(* CODESYS project retain.paras.190613.2.project

Project tree, tasks and I/O mapping:
  MIC7001 : Changsha Xiangji-ARM Cortex A9(xilinx zynq7000)-linux, Changsha Xiangji Hiden Technology Co.Ltd, version 3.5.10.40
    application Application
      libraries: Standard, * (System); CAA File, * (CAA Technical Workgroup); CAA Types Extern, * (CAA Technical Workgroup); CAA Callback Extern, * (CAA Technical Workgroup); SysMem, * (System); Util, 3.5.11.0 (System); SysFile, 3.5.9.0 (System); SysTypes Interfaces, * (System); CAN API, 1.0.0.3 (3S - Smart Software Solutions GmbH); SysTime, * (System); CAA DTUtil Extern, 3.5.12.0 (CAA Technical Workgroup); CAA SerialCom, 3.5.12.0 (CAA Technical Workgroup); cyber gpio, 3.5.10.40 (cyber); AC_DataLog, 3.5.13.0 (3S - Smart Software Solutions GmbH)
      task MainTask (cyclic, interval 20 ms, priority 15) calls prg_main
      task task_retain (cyclic, interval 200 ms, priority 19) calls prg_retain_paras
      global variables GVL
      retain_para/
        data type DUT_PARA_DINT
        data type DUT_PARA_REAL
        function block FB_PARA_DINT [ST]: wr_all, clear_all, rd_all, chk_chg
        function block FB_PARA_REAL [ST]: clear_all, wr_all, rd_all, chk_chg
        program prg_retain_paras [ST]
      program prg_main [ST]
    SoftMotion General Axis Pool
  text list GlobalTextList
*)

// MIC7001/Application/retain_para/DUT_PARA_DINT
TYPE DUT_PARA_DINT :
STRUCT
	num:UINT := 64;  //可根据需要设置总数量，最后一个为校验和，不可用
	para:ARRAY[0..64] OF DINT;  //三行中的总数量需要严格一致,位置0 用于存放魔法数字
	old_val:ARRAY[0..64] OF DINT; //三行中的总数量需要严格一致,位置0 用于存放魔法数字
	filename :STRING := '/userapp/mic_dint.txt';  
END_STRUCT
END_TYPE

// MIC7001/Application/retain_para/DUT_PARA_REAL
TYPE DUT_PARA_REAL :
STRUCT
	num:UINT := 256; //可根据需要设置总数量，最后一个为校验和，不可用
	para:ARRAY[0..256] OF REAL;  //三行中的总数量需要严格一致,位置0 用于存放魔法数字
	old_val:ARRAY[0..256] OF REAL; //三行中的总数量需要严格一致,位置0 用于存放魔法数字
	filename :STRING := '/userapp/mic_real.txt';  
END_STRUCT
END_TYPE

// MIC7001/Application/GVL
VAR_GLOBAL
	user_para_01: DINT := 1234;
	user_para_02: DINT := 3323;
	user_para_03: DINT := 4322;
END_VAR

// MIC7001/Application/prg_main
PROGRAM prg_main
VAR
	cntr :dint := 0;
END_VAR


cntr := cntr + 1;

IF cntr > 100 THEN
	gvl.user_para_01 := gvl.user_para_01 + 1;
	gvl.user_para_02 := gvl.user_para_02 + 2;
	
	gvl.user_para_03 := gvl.user_para_03 + 0;
	
	cntr := 0;
END_IF

END_PROGRAM

// MIC7001/Application/retain_para/prg_retain_paras
PROGRAM prg_retain_paras
VAR
	data_stat:UINT := 0;
    myRetainMigicNumber:DINT := 1324904337;  //本机型的魔法数字，必须修改，越随机越好
END_VAR

VAR_INPUT
	para_dint:DUT_PARA_DINT;
	retain_dint:FB_PARA_DINT;
END_VAR

//整数参数掉电存储例程

// (1) 拷贝本工程内的 parameters 目录到用户自己的工程;
// (2) 将其中的prg_retain_paras 程序拷贝到 某一个任务中；
// (3) 使用自己定义的变量替换掉 gvl.user_para_01,   gvl.user_para_02 和 gvl.user_para_03, 并更改本程序中对应的变量
// (4) 如果需要保存更多的变量，可仿照本例增加变量（默认支持64个） 

retain_dint(enable := TRUE, pPara := ADR(para_dint));

CASE data_stat OF
0:
	IF retain_dint.zero OR para_dint.para[0] <> myRetainMigicNumber  THEN   //数据为空或者魔法数字错误，恢复初始值
		para_dint.para[0] := myRetainMigicNumber;
		para_dint.para[1] := gvl.user_para_01;
		para_dint.para[2] := gvl.user_para_02;
		para_dint.para[3] := gvl.user_para_03;
		//para_dint.para[4] := gvl.user_para_04;  
		//可在此处添加新的用户变量
	ELSE
		gvl.user_para_01 := para_dint.para[1];
		gvl.user_para_02 := para_dint.para[2];
		gvl.user_para_03 := para_dint.para[3];
		//gvl.user_para_04 := para_dint.para[4];  
		//可在此处添加新的用户变量
		
		data_stat := 10;
	END_IF
10:
	para_dint.para[1] := gvl.user_para_01;
	para_dint.para[2] := gvl.user_para_02;
	para_dint.para[3] := gvl.user_para_03;
	//para_dint.para[4] := gvl.user_para_04;  
	//可在此处添加新的用户变量
	
END_CASE

END_PROGRAM

// MIC7001/Application/retain_para/FB_PARA_DINT
FUNCTION_BLOCK FB_PARA_DINT
VAR_INPUT
	enable:BOOL := FALSE;
	clear:BOOL := FALSE;
	pPara:POINTER TO DUT_PARA_DINT;
END_VAR

VAR_OUTPUT
	ok:BOOL := FALSE;
	zero:BOOL := FALSE;
END_VAR

VAR
	hFile: RTS_IEC_HANDLE := 0;
	sync:BOOL := FALSE;  
	stat:UINT:= 0;
	
	i :UINT;
END_VAR


IF NOT enable OR pPara^.num < 1 THEN
	stat := 0;
	RETURN;
END_IF

CASE stat OF
	0:  //init
		IF rd_all(pPara^.filename)	THEN 
			zero := FALSE;
			ok := TRUE;
			stat := 10;
		ELSE
			clear_all();
			IF wr_all(pPara^.filename) THEN
				zero := TRUE;
				ok := FALSE;
				stat := 10;
			END_IF
		END_IF
	
	10: // normal
		IF chk_chg() THEN
			ok := FALSE;
			IF wr_all(pPara^.filename) THEN
				ok := TRUE;
				zero := FALSE;
			END_IF
		END_IF	
		
		IF clear THEN
			clear_all();
			IF wr_all(pPara^.filename) THEN
				zero := TRUE;
				ok := FALSE;
			END_IF
		END_IF
END_CASE

METHOD wr_all : bool
VAR_INPUT
	filename:STRING(256);
END_VAR

VAR
	iNumber:INT;
	udiByteWrite:LWORD;
	udiPos:UDINT;
	udiOpenError: RTS_IEC_RESULT;
	udiWriteError: RTS_IEC_RESULT;
	str_size:DWORD;
	str: STRING(255);
	check_sum: DINT;
END_VAR
wr_all := FALSE;
hFile := sysfileopen(szFile := filename, am := sysfile.AM_WRITE, pResult := ADR(udiOpenError));
IF hFile = RTS_INVALID_HANDLE THEN
	RETURN;
END_IF

udiPos := SysFileSetPos(hFile:=hFile, ulOffset := 0);

check_sum := 0;
str:= ANY_TO_STRING('');
FOR i := 0 TO pPara^.num DO
	IF i = pPara^.num THEN  //the last val, check_sum
		pPara^.para[i] := check_sum;
	ELSE
		check_sum := check_sum + pPara^.para[i];
	END_IF
	str := concat(str, ANY_TO_STRING(pPara^.para[i]));
	str := concat(str, ANY_TO_STRING('$N'));
	str_size := ANY_TO_DWORD(len(str));
	IF str_size > 200 THEN
		udiByteWrite := sysfile.SysFileWrite(hFile := hFile,pbyBuffer := ADR(str),ulSize := str_size, pResult := ADR(udiWriteError));
		IF udiByteWrite = str_size THEN
			str := '';
		END_IF
	END_IF	
END_FOR
udiByteWrite := sysfile.SysFileWrite(hFile := hFile,pbyBuffer := ADR(str),ulSize := str_size, pResult := ADR(udiWriteError));
	
IF udiByteWrite <> str_size THEN
	sysfile.SysFileClose(hFile);
	RETURN;
END_IF
sysfile.SysFileClose(hFile);

	
FOR i := 0 TO pPara^.num DO
	pPara^.old_val[i] := pPara^.para[i];
END_FOR

hFile := 0;

wr_all := TRUE;
END_METHOD

METHOD clear_all : bool
VAR_INPUT
	
END_VAR
FOR i := 0 TO pPara^.num DO
	pPara^.para[i] := 0;
	pPara^.old_val[i] := 0;
END_FOR

clear_all := TRUE;
END_METHOD

METHOD rd_all : bool
VAR_INPUT
	filename:STRING(256);
END_VAR

VAR
	iNumber:INT;
	udiByteRead:LWORD;
	udiPos:UDINT;
	udiOpenError: RTS_IEC_RESULT;
	udiReadError: RTS_IEC_RESULT;
	str: STRING(255);
	ulOffset:DWORD;
	batch: BOOL;
	check_sum: DINT;
END_VAR
rd_all := FALSE;

hFile := sysfileopen(szFile := filename, am := sysfile.AM_READ, pResult:= ADR(udiOpenError));
IF hFile = RTS_INVALID_HANDLE THEN
	RETURN;
END_IF

ulOffset := 0;
batch := TRUE;

check_sum := 0;
FOR i := 0 TO pPara^.num DO
	IF udiByteRead < 50 AND batch THEN
		udiPos := SysFileSetPos(hFile:=hFile, ulOffset := ulOffset);
		udiByteRead := sysfile.SysFileRead(hfile := hFile,pbyBuffer := ADR(str), ulSize := 255 , pResult := ADR(udiReadError));
		IF udiByteRead < 255 THEN
			batch := FALSE;
		END_IF
	END_IF
	IF udiByteRead < 1 THEN  //读取失败
		sysfile.SysFileClose(hFile := hFile);
		RETURN;
	END_IF

	iNumber := find(str, '$N');
	IF iNumber < 2 THEN
		sysfile.SysFileClose(hFile := hFile);
		RETURN;
	END_IF
	
	pPara^.para[i] := STRING_TO_DINT(left(str,iNumber-1));
	str := delete(str, iNumber,1);
	pPara^.old_val[i] := pPara^.para[i];
	
	udiByteRead := udiByteRead - ANY_TO_LWORD(iNumber);
	ulOffset := ulOffset + ANY_TO_DWORD(iNumber);

	IF i = pPara^.num THEN
		IF check_sum <> pPara^.para[i] THEN
			RETURN;  //error
		END_IF
	ELSE
		check_sum := check_sum + pPara^.para[i];
	END_IF
END_FOR

sysfile.SysFileClose(hFile := hFile);
rd_all := TRUE;
END_METHOD

METHOD chk_chg : bool
VAR_INPUT
END_VAR

VAR
	i :UINT;
END_VAR
chk_chg := TRUE;

FOR i := 0 TO pPara^.num  DO
	IF pPara^.para[i] <> pPara^.old_val[i] THEN
		RETURN;
	END_IF
END_FOR

chk_chg := FALSE;
END_METHOD

END_FUNCTION_BLOCK

// MIC7001/Application/retain_para/FB_PARA_REAL
FUNCTION_BLOCK FB_PARA_REAL
VAR_INPUT
	enable:BOOL := FALSE;
	clear:BOOL := FALSE;
	pPara:POINTER TO DUT_PARA_REAL;
END_VAR

VAR_OUTPUT
	ok:BOOL := FALSE;
	zero:BOOL := FALSE;
END_VAR

VAR
	hFile: RTS_IEC_HANDLE := 0;
	sync:BOOL := FALSE;  
	stat:UINT:= 0;
	
	i :UINT;
	str:STRING(1024);
END_VAR


IF NOT enable OR pPara^.num < 1 THEN
	stat := 0;
	RETURN;
END_IF

CASE stat OF
	0:  //init
		IF rd_all(pPara^.filename)	THEN 
			zero := FALSE;
			stat := 10;
		ELSE
			clear_all();
			IF wr_all(pPara^.filename) THEN
				zero := TRUE;
				stat := 10;
			END_IF
		END_IF
	
	10: // normal
		IF chk_chg() THEN
			ok := FALSE;
			IF wr_all(pPara^.filename) THEN
				ok := TRUE;
				zero := FALSE;
			END_IF
		END_IF	
		
		IF clear THEN
			clear_all();
			IF wr_all(pPara^.filename) THEN
				zero := TRUE;
			END_IF
		END_IF
END_CASE

METHOD clear_all : bool
VAR_INPUT
	
END_VAR
FOR i := 0 TO pPara^.num DO
	pPara^.para[i] := 0.0;
	pPara^.old_val[i] := 0.0;
END_FOR

clear_all := TRUE;
END_METHOD

METHOD wr_all : bool
VAR_INPUT
	filename:STRING(256);
END_VAR

VAR
	iNumber:INT;
	udiByteWrite:LWORD;
	udiPos:UDINT;
	udiOpenError: RTS_IEC_RESULT;
	udiWriteError: RTS_IEC_RESULT;
	str_size:DWORD;
	check_sum: REAL;
END_VAR
wr_all := FALSE;
hFile := sysfileopen(szFile := filename, am := sysfile.AM_WRITE, pResult := ADR(udiOpenError));
IF hFile = RTS_INVALID_HANDLE THEN
	RETURN;
END_IF

udiPos := SysFileSetPos(hFile:=hFile, ulOffset := 0);

check_sum := 0.0;
str:= ANY_TO_STRING('');
FOR i := 0 TO pPara^.num DO
	IF i = pPara^.num THEN  //the last val, check_sum
		pPara^.para[i] := check_sum;
	ELSE
		check_sum := check_sum + pPara^.para[i];
	END_IF	
	str := concat(str, ANY_TO_STRING(pPara^.para[i]));
	str := concat(str, ANY_TO_STRING('$N'));
	str_size := ANY_TO_DWORD(len(str));
	IF str_size > 200 THEN
		udiByteWrite := sysfile.SysFileWrite(hFile := hFile,pbyBuffer := ADR(str),ulSize := str_size, pResult := ADR(udiWriteError));
		IF udiByteWrite = str_size THEN
			str := '';
		END_IF
	END_IF	
END_FOR
udiByteWrite := sysfile.SysFileWrite(hFile := hFile,pbyBuffer := ADR(str),ulSize := str_size, pResult := ADR(udiWriteError));
	
IF udiByteWrite <> str_size THEN
	sysfile.SysFileClose(hFile);
	RETURN;
END_IF
sysfile.SysFileClose(hFile);

	
FOR i := 0 TO pPara^.num DO
	pPara^.old_val[i] := pPara^.para[i];
END_FOR

hFile := 0;

wr_all := TRUE;
END_METHOD

METHOD rd_all : bool
VAR_INPUT
	filename:STRING(256);
END_VAR

VAR
	iNumber:INT;
	udiByteRead:LWORD;
	udiPos:UDINT;
	udiOpenError: RTS_IEC_RESULT;
	udiReadError: RTS_IEC_RESULT;
	str: STRING(255);
	ulOffset:DWORD;
	batch: BOOL;
	check_sum :REAL;
END_VAR
rd_all := FALSE;

hFile := sysfileopen(szFile := filename, am := sysfile.AM_READ, pResult:= ADR(udiOpenError));
IF hFile = RTS_INVALID_HANDLE THEN
	RETURN;
END_IF

ulOffset := 0;
batch := TRUE;

check_sum := 0.0;
FOR i := 0 TO pPara^.num DO
	IF udiByteRead < 50 AND batch THEN
		udiPos := SysFileSetPos(hFile:=hFile, ulOffset := ulOffset);
		udiByteRead := sysfile.SysFileRead(hfile := hFile,pbyBuffer := ADR(str), ulSize := 255 , pResult := ADR(udiReadError));
		IF udiByteRead < 255 THEN
			batch := FALSE;
		END_IF
	END_IF
	IF udiByteRead < 1 THEN  //读取失败
		sysfile.SysFileClose(hFile := hFile);
		RETURN;
	END_IF

	iNumber := find(str, '$N');
	IF iNumber < 2 THEN
		sysfile.SysFileClose(hFile := hFile);
		RETURN;
	END_IF
	
	pPara^.para[i] := STRING_TO_REAL(left(str,iNumber-1));
	str := delete(str, iNumber,1);
	pPara^.old_val[i] := pPara^.para[i];
	
	udiByteRead := udiByteRead - ANY_TO_LWORD(iNumber);
	ulOffset := ulOffset + ANY_TO_DWORD(iNumber);

	IF i = pPara^.num THEN
		IF ABS(check_sum-pPara^.para[i]) > 0.01 THEN
			RETURN;  //error
		END_IF
	ELSE
		check_sum := check_sum + pPara^.para[i];
	END_IF
END_FOR

sysfile.SysFileClose(hFile := hFile);
rd_all := TRUE;
END_METHOD

METHOD chk_chg : bool
VAR_INPUT
END_VAR

VAR
	i :UINT;
END_VAR
chk_chg := TRUE;

FOR i := 0 TO pPara^.num  DO
	IF pPara^.para[i] <> pPara^.old_val[i] THEN
		RETURN;
	END_IF
END_FOR

chk_chg := FALSE;
END_METHOD

END_FUNCTION_BLOCK
